// TIA Portal V20 export
DATA_BLOCK "Param"   // DB352
{ S7_Optimized_Access := 'FALSE' }
// stored: AutoNumber false
   VAR RETAIN
      Plc : "TypeHeaderPlc";   // Header Plc
      Rd : Struct
         watchdog : Int := 0;   // watchdog
         adjHousingOff : Int := 0;   // adjustment scanner housing off (only manual movement possible ) [On/Off]
         adjTopOff : Int := 0;   // adjustment camera top off (only manual movement possible ) [On/Off]
         adjLeftOff : Int := 0;   // adjustment camera left off (only manual movement possible ) [On/Off]
         adjRightOff : Int := 0;   // adjustment camera right off (only manual movement possible ) [On/Off]
         adjLaserTopLeftStepMotOff : Int;   // adjustment laser top left off (only manual movement possible ) [On/Off]
         adjLaserTopRightStepMotOff : Int;   // adjustment laser top right off (only manual movement possible ) [On/Off]
         adjLaserLeftTopStepMotOff : Int;   // adjustment laser left top off (only manual movement possible ) [On/Off]
         adjLaserLeftBottomStepMotOff : Int;   // adjustment laser left bottom off (only manual movement possible ) [On/Off]
         adjLaserRightTopStepMotOff : Int;   // adjustment laser right top off (only manual movement possible ) [On/Off]
         adjLaserRightBottomStepMotOff : Int;   // adjustment laser right bottom off (only manual movement possible ) [On/Off]
         param1 : Int;
         param2 : Int;
         param3 : Int;
         param4 : Int;
         air1Off : Int := 0;   // air conditioner 1 scannerhousing visual measurement [On/Off]
         air2Off : Int := 0;   // air conditioner 2 scannerhousing visual measurement [On/Off]
         airXrayOff : Int := 0;   // air conditioner scannerhousing x-ray measurement [On/Off]
         airDehOff : Int := 0;   // air dehumidifier
         param5 : Int := 0;
         param6 : Int := 0;
         blowOffImpuls : Int := 400;   // blow off impulse [ms]
         blowOffIbreak : Int := 400;   // blow off minimum break to start new cycle [ms]
         blowOffintervall : Int := 120;   // blow off interval if no board pass [s]
         param10 : Int := 0;
         air1Active : Int := 1;   // air conditioner 1 scannerhousing visual measurement active [On/Off]
         air1InputNo : Int := 0;   // air conditioner 1 scannerhousing visual measurement input normal [On/Off]
         air2Active : Int := 0;   // air conditioner 2 scannerhousing visual measurement active [On/Off]
         air2InputNo : Int := 0;   // air conditioner 2 scannerhousing visual measurement input normal [On/Off]
         airXrayActive : Int := 1;   // air conditioner scannerhousing x-ray measurement active [On/Off]
         airXrayInputNo : Int := 0;   // air conditioner scannerhousing x-ray measurement input normal [On/Off]
         airDehActive : Int := 0;   // air dehumidifier active [On/Off]
         airDehInputNo : Int := 0;   // air dehumidifier input normal open [On/Off]
         param11 : Int := 0;
         blowOffintervallOff : Int := 600;   // blow off interval if no board pass switches off after this time [s]
         blowOffDelayStartBottom : Int := 0;   // blow off delay start for valve bottom [ms]
         blowOffDelayStartLeft : Int := 0;   // blow off delay start for valve left [ms]
         blowOffDelayStartRight : Int := 0;   // blow off delay start for valve right [ms]
         blowOffDelayStartXray : Int := 0;   // blow off delay start for valve xray [ms]
         blowOffImpulsBottom : Int := 400;   // blow off impulse for valve bottom [ms]
         blowOffImpulsLeft : Int := 400;   // blow off impulse for valve left [ms]
         blowOffImpulsRight : Int := 400;   // blow off impulse for valve right [ms]
         blowOffImpulsXray : Int := 400;   // blow off impulse for valve xray [ms]
         ParamRes : Array[1..58] of Int;
      END_STRUCT;
   END_VAR
BEGIN
   Plc.conActive := FALSE;
   Plc.err := FALSE;
   Plc.errWd := FALSE;
   Plc.errSd := FALSE;
   Plc.errRd := FALSE;
   Plc.bit05 := FALSE;
   Plc.bit06 := FALSE;
   Plc.bit07 := FALSE;
   Plc.sdBusy := FALSE;
   Plc.sdDone := FALSE;
   Plc.rdBusy := FALSE;
   Plc.rdDone := FALSE;
   Plc.sdOverload := FALSE;
   Plc.statistic := FALSE;
   Plc.bit16 := FALSE;
   Plc.bit17 := FALSE;
   Plc.sdState := 16#0000;
   Plc.sdLastErrState := 16#0000;
   Plc.sdLenght := 0;
   Plc.sdCps := 0;
   Plc.rdState := 16#0000;
   Plc.rdLastErrState := 16#0000;
   Plc.rdLenght := 0;
   Plc.rdCps := 0;
   Plc.in18 := 0;
   Rd.ParamRes[1..50] := 0;
END_DATA_BLOCK
